{attribute 'qualified_only'}
{attribute 'strict'}
TYPE E_State :
(
	OFF := 0,
	IDLE := 1,
	START_WATER_FLOW := 2,
	RUNNING := 3,
	COOLDOWN := 4,
    ERROR := 5
);
END_TYPE

(* stored: Version 1.1.0.1
   DUT E_State: Id {94a8806a-5b5b-4337-85e8-4f8b07c6bd5b} *)
